FUNCTION_BLOCK xPPU_RFC
VAR_INPUT
	i_error: POINTER TO ErrorManager;
	i_process: POINTER TO ProcessManager;
	i_state: POINTER TO StateTracker;
END_VAR
VAR
	m_emptyParams: ParameterSet;
	m_subRes: EOperationResult;
END_VAR

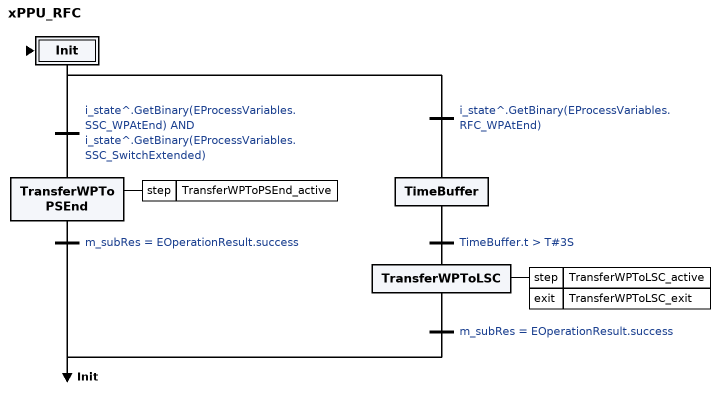
INITIAL_STEP Init:
END_STEP
TRANSITION FROM Init TO TransferWPToPSEnd
    := i_state^.GetBinary(EProcessVariables.SSC_WPAtEnd) AND i_state^.GetBinary(EProcessVariables.SSC_SwitchExtended);
END_TRANSITION
STEP TransferWPToPSEnd:
    TransferWPToPSEnd_active(N);  // step action
END_STEP
TRANSITION FROM TransferWPToPSEnd TO Init
    := m_subRes = EOperationResult.success;
END_TRANSITION
TRANSITION FROM Init TO TimeBuffer
    := i_state^.GetBinary(EProcessVariables.RFC_WPAtEnd);
END_TRANSITION
STEP TimeBuffer:
END_STEP
TRANSITION FROM TimeBuffer TO TransferWPToLSC
    := TimeBuffer.t > T#3S;
END_TRANSITION
STEP TransferWPToLSC:
    TransferWPToLSC_active(N);  // step action
    TransferWPToLSC_exit(P0);  // exit action
END_STEP
TRANSITION FROM TransferWPToLSC TO Init
    := m_subRes = EOperationResult.success;
END_TRANSITION

ACTION TransferWPToLSC_active:
m_subRes := i_process^.Execute(
	EBehaviorType.control_primitive,
	EPrimitives.RFC_TransferWorkpieceTo_LSC,
	m_emptyParams);
END_ACTION

ACTION TransferWPToLSC_exit:
i_state^.ShiftProduct(EProducts.RFC_product1, EProducts.LSC_product);
IF i_state^.GetBinary(EProcessVariables.RFC_WPAtEnd) THEN
	i_state^.ShiftProduct(EProducts.RFC_product2, EProducts.RFC_product1);
END_IF
END_ACTION

ACTION TransferWPToPSEnd_active:
m_subRes := i_process^.Execute(
	EBehaviorType.control_primitive,
	EPrimitives.RFC_TransferWorkpieceTo_PSEnd,
	m_emptyParams);
END_ACTION

END_FUNCTION_BLOCK

(* stored: Version 1.1.0.1, ProductVersion 3.1.4024.4
   POU xPPU_RFC: Id {d90f6f73-9cc6-49aa-95fa-83b2098b3cd4}, SpecialFunc None
   Action TransferWPToLSC_active: Id {06822a62-8370-4767-a20c-06a31bc41e8d}
   Action TransferWPToLSC_exit: Id {47333ae5-1a92-4122-ac22-bb58dd1f2d05}
   Action TransferWPToPSEnd_active: Id {7486f9de-223c-4795-a1d2-77997eb33773} *)
